TYPE st_diagFBBits :ARRAY[0..15] OF BOOL;
END_TYPE

(* stored: Version 1.1.0.1, ProductVersion 3.1.4024.12
   DUT st_diagFBBits: Id {51771b6c-fb7a-440c-9cab-f62079bacb1f} *)
